{attribute 'GeneratedUsingTerminal: EP2328-1061-0016'}
{attribute addProperty BoxType "EP2328-1061-0016"}
{attribute addProperty Id "DI_X01_Pin4_InputAT %I*DI_X01_Pin4_Input_830843C11DI_X01_Pin2_InputAT %I*DI_X01_Pin2_Input_830843C11DI_X02_Pin4_InputAT %I*DI_X02_Pin4_Input_830843C11DI_X02_Pin2_InputAT %I*DI_X02_Pin2_Input_830843C11DO_X03_Pin4_OutputAT %Q*DO_X03_Pin4_Output_42CA91F71DO_X03_Pin2_OutputAT %Q*DO_X03_Pin2_Output_42CA91F71DO_X04_Pin4_OutputAT %Q*DO_X04_Pin4_Output_42CA91F71DO_X04_Pin2_OutputAT %Q*DO_X04_Pin2_Output_42CA91F71WcStateAT %I*WcState_9091E0EB2InfoDataAT %I*InfoData_6F19DB2B2"}
{attribute addProperty CRC "4134329783"}
{attribute addProperty Size "12"}
TYPE EP2328_F66CDDB7 EXTENDS EtcSlaveTerminalBase_947E5A46 :
STRUCT
	{attribute addProperty Name "DI_X01_Pin4_Input"}
	DI_X01_Pin4_Input : DI_X01_Pin4_Input_830843C1;
	{attribute addProperty Name "DI_X01_Pin2_Input"}
	DI_X01_Pin2_Input : DI_X01_Pin2_Input_830843C1;
	{attribute addProperty Name "DI_X02_Pin4_Input"}
	DI_X02_Pin4_Input : DI_X02_Pin4_Input_830843C1;
	{attribute addProperty Name "DI_X02_Pin2_Input"}
	DI_X02_Pin2_Input : DI_X02_Pin2_Input_830843C1;
	{attribute addProperty Name "DO_X03_Pin4_Output"}
	DO_X03_Pin4_Output : DO_X03_Pin4_Output_42CA91F7;
	{attribute addProperty Name "DO_X03_Pin2_Output"}
	DO_X03_Pin2_Output : DO_X03_Pin2_Output_42CA91F7;
	{attribute addProperty Name "DO_X04_Pin4_Output"}
	DO_X04_Pin4_Output : DO_X04_Pin4_Output_42CA91F7;
	{attribute addProperty Name "DO_X04_Pin2_Output"}
	DO_X04_Pin2_Output : DO_X04_Pin2_Output_42CA91F7;
	{attribute addProperty Name "WcState"}
	WcState : WcState_9091E0EB;
	{attribute addProperty Name "InfoData"}
	InfoData : InfoData_6F19DB2B;
END_STRUCT
END_TYPE

(* stored: Version 1.2.0.0, ProductVersion 3.1.4024.9
   DUT EP2328_F66CDDB7: Id {9da6db88-b184-454c-84af-52e85303dcf8} *)
